TYPE ST_Netcontactor_get :
STRUCT
	e_NetConState					: eNetcontactorState;
	b_SyncCloseCommand				: BOOL;
	b_NetConFb						: BOOL;
	b_NetcontRightFb				: BOOL;
	b_NetcontLeftFb					: BOOL;
	events							: ST_Netcontactor_events;
END_STRUCT
END_TYPE

(* stored: Version 1.1.0.1, ProductVersion 3.1.4026.18
   DUT ST_Netcontactor_get: Id {9f29cdd3-c248-455e-a8be-dde6b5050d72} *)
